FUNCTION INTERNAL F_SetMessageValue : E_WriterErrorCode
VAR_INPUT
	anyValue : T_ANY;
	iMessage : I_Message;
END_VAR
VAR
	anyMessage : T_ANY;
END_VAR

IF iMessage = NULL THEN
	 F_SetMessageValue := E_WriterErrorCode.InternalError;
	 RETURN;
END_IF;

anyMessage := iMessage.MessageValue;
IF anyValue.diSize <> anyMessage.diSize THEN
	 F_SetMessageValue := E_WriterErrorCode.InternalError;
	 RETURN;
END_IF;
 
MEMCPY(destAddr:= anyMessage.pValue, srcAddr:= anyValue.pValue, n:= TO_UDINT(anyValue.diSize));

END_FUNCTION

(* stored: Version 1.1.0.1
   POU F_SetMessageValue: Id {4930023b-9dbb-4d90-957d-7d922826a85b}, SpecialFunc None *)
